INTERFACE I_TankFill

METHOD Close : BOOL
VAR_INPUT
END_VAR
END_METHOD

PROPERTY IsClose : bool
GET
END_GET
END_PROPERTY

PROPERTY IsOpen : bool
GET
END_GET
END_PROPERTY

METHOD Open : BOOL
VAR_INPUT
END_VAR
END_METHOD

END_INTERFACE

(* stored: Version 1.1.0.1, ProductVersion 3.1.4024.12
   Itf I_TankFill: Id {0e48e970-fee3-4f32-8378-3931954799d0}
   Method Close: Id {6fb8ca09-7b6a-4324-9a9a-9e4d83106e22}
   Property IsClose: Id {17b38770-f8d0-46e2-b56a-ce5e295c4401}
   Get Get: Id {21ad2a2d-918d-4451-9142-497d571761a3}
   Property IsOpen: Id {15d05cd5-24af-441e-a9c5-4a6db77c2c5b}
   Get Get: Id {2e4102c4-8500-4871-a7a5-aa77cadc09e3}
   Method Open: Id {b28b4c71-5590-4f2d-8489-25b460fb5848} *)
